Omron CX-Programmer project NewProject (CX-Programmer 9.73)

# PLC NewPLC1: CP1E E30

## Global symbols (name address type ; comment)
0.00 BOOL  ; A
0.01 BOOL  ; B
0.02 BOOL  ; C
0.03 BOOL  ; D
0.04 BOOL  ; E
0.05 BOOL  ; F
100.00 BOOL  ; G1 naik
100.01 BOOL  ; G1 turun
100.02 BOOL  ; G2 naik
100.03 BOOL  ; G2 turun
100.04 BOOL  ; G3 naik
100.05 BOOL  ; G3 turun
100.06 BOOL  ; V1 penuh
100.07 BOOL  ; V2 penuh
10.00 BOOL  ; set G1 turun
10.01 BOOL  ; set G2 turun
10.02 BOOL  ; set G3 turun
11.00 BOOL  ; NOP
D1 CHANNEL  ; data V1
D2 CHANNEL  ; data V2
T000 BOOL  ; delay G1 naik
T001 BOOL  ; delay set G1 turun
T002 BOOL  ; delay G1 turun
T004 BOOL  ; delay G2 naik
T005 BOOL  ; delay set G2 turun
T006 BOOL  ; delay G2 turun
T007 BOOL  ; delay G3 naik
T008 BOOL  ; delay set G3 turun
T009 BOOL  ; delay G3 turun
W0.01 BOOL  ; M.V1
W0.02 BOOL  ; M.V2

## Program NewProgram1 (cyclic task 0)

### Section PROGRAM

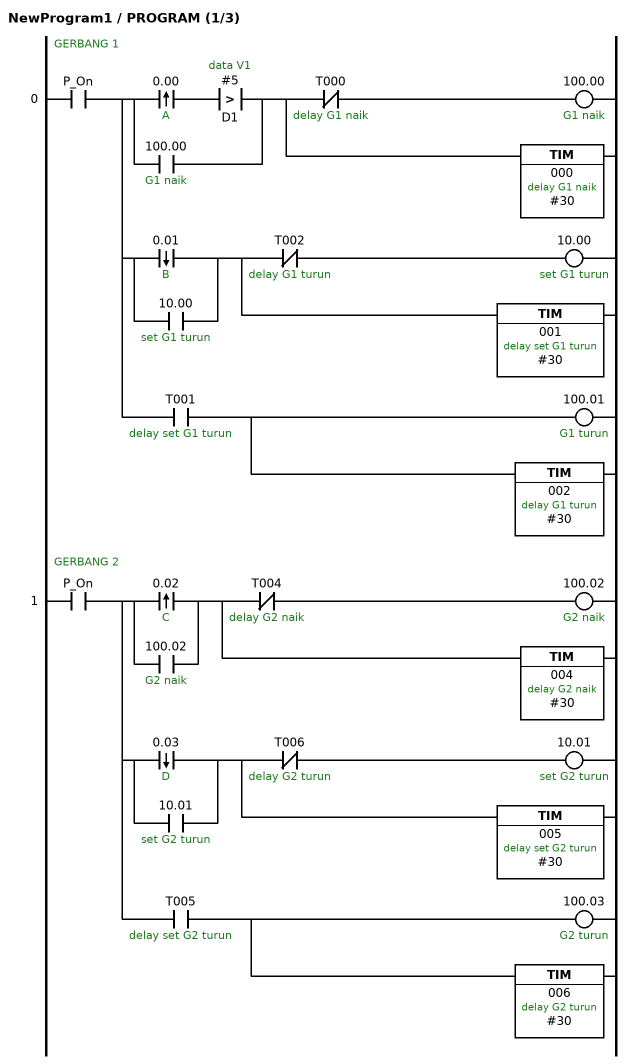
; rung 0: GERBANG 1
LD P_On
OUT TR0
@LD 0.00  ; A
AND>(320) #5 D1  ; data V1
OR 100.00  ; G1 naik
ANDLD
OUT TR1
ANDNOT T000  ; delay G1 naik
OUT 100.00  ; G1 naik
LD TR1
TIM 000 #30  ; delay G1 naik
LD TR0
%LD 0.01  ; B
OR 10.00  ; set G1 turun
ANDLD
OUT TR1
ANDNOT T002  ; delay G1 turun
OUT 10.00  ; set G1 turun
LD TR1
TIM 001 #30  ; delay set G1 turun
LD TR0
AND T001  ; delay set G1 turun
OUT 100.01  ; G1 turun
TIM 002 #30  ; delay G1 turun
; rung 1: GERBANG 2
LD P_On
OUT TR0
@LD 0.02  ; C
OR 100.02  ; G2 naik
ANDLD
OUT TR1
ANDNOT T004  ; delay G2 naik
OUT 100.02  ; G2 naik
LD TR1
TIM 004 #30  ; delay G2 naik
LD TR0
%LD 0.03  ; D
OR 10.01  ; set G2 turun
ANDLD
OUT TR1
ANDNOT T006  ; delay G2 turun
OUT 10.01  ; set G2 turun
LD TR1
TIM 005 #30  ; delay set G2 turun
LD TR0
AND T005  ; delay set G2 turun
OUT 100.03  ; G2 turun
TIM 006 #30  ; delay G2 turun

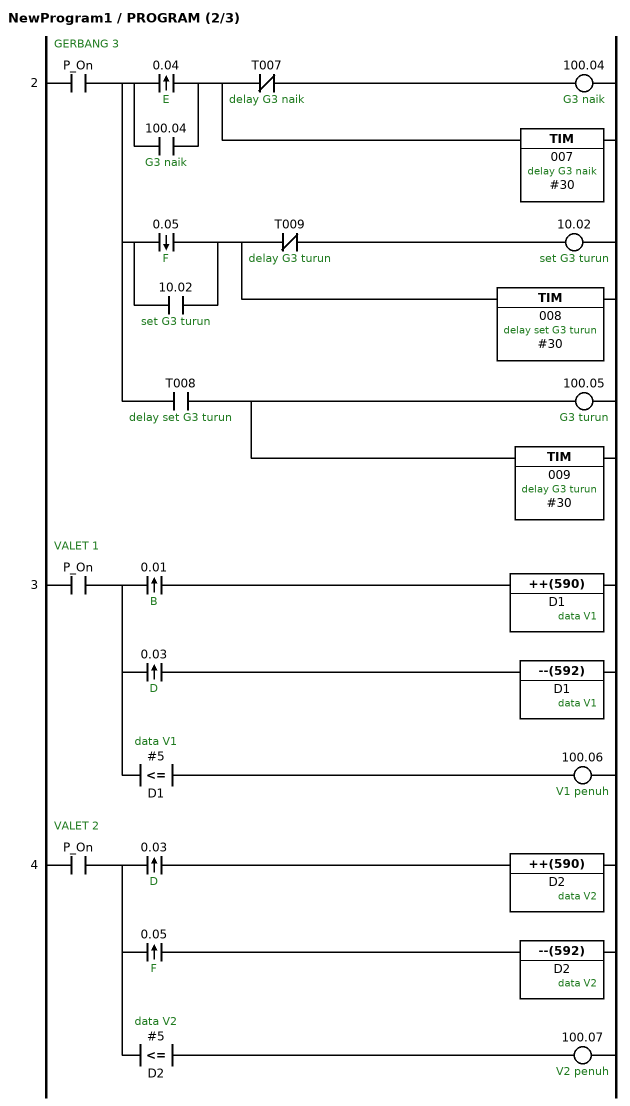
; rung 2: GERBANG 3
LD P_On
OUT TR0
@LD 0.04  ; E
OR 100.04  ; G3 naik
ANDLD
OUT TR1
ANDNOT T007  ; delay G3 naik
OUT 100.04  ; G3 naik
LD TR1
TIM 007 #30  ; delay G3 naik
LD TR0
%LD 0.05  ; F
OR 10.02  ; set G3 turun
ANDLD
OUT TR1
ANDNOT T009  ; delay G3 turun
OUT 10.02  ; set G3 turun
LD TR1
TIM 008 #30  ; delay set G3 turun
LD TR0
AND T008  ; delay set G3 turun
OUT 100.05  ; G3 turun
TIM 009 #30  ; delay G3 turun
; rung 3: VALET 1
LD P_On
OUT TR0
@AND 0.01  ; B
++(590) D1  ; data V1
LD TR0
@AND 0.03  ; D
--(592) D1  ; data V1
LD TR0
AND<=(315) #5 D1  ; data V1
OUT 100.06  ; V1 penuh
; rung 4: VALET 2
LD P_On
OUT TR0
@AND 0.03  ; D
++(590) D2  ; data V2
LD TR0
@AND 0.05  ; F
--(592) D2  ; data V2
LD TR0
AND<=(315) #5 D2  ; data V2
OUT 100.07  ; V2 penuh

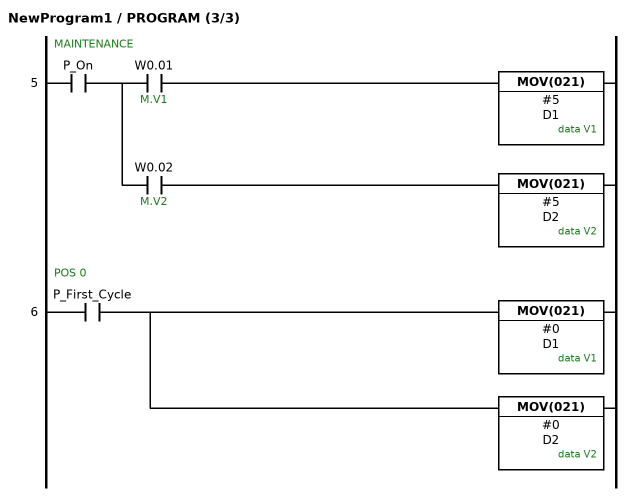
; rung 5: MAINTENANCE
LD P_On
OUT TR0
AND W0.01  ; M.V1
MOV(021) #5 D1  ; data V1
LD TR0
AND W0.02  ; M.V2
MOV(021) #5 D2  ; data V2
; rung 6: POS 0
LD P_First_Cycle
MOV(021) #0 D1  ; data V1
MOV(021) #0 D2  ; data V2

### Section IN_OUT

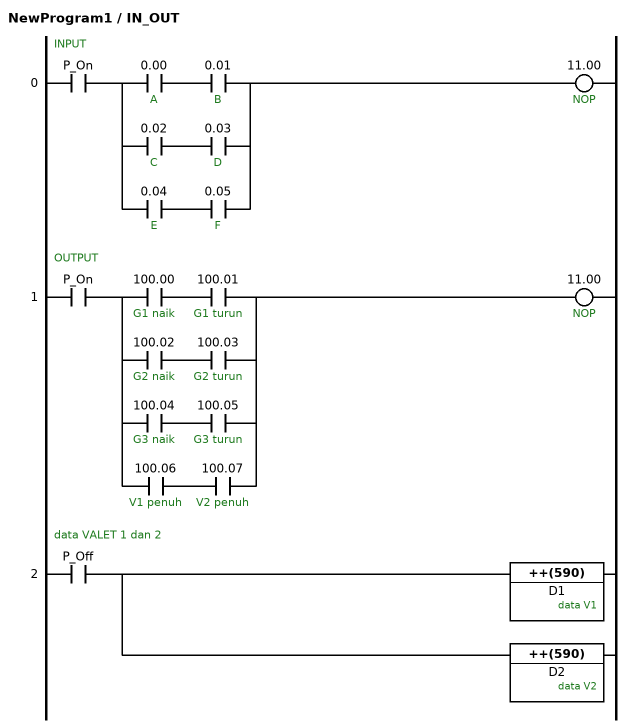
; rung 0: INPUT
LD P_On
LD 0.00  ; A
AND 0.01  ; B
LD 0.02  ; C
AND 0.03  ; D
ORLD
LD 0.04  ; E
AND 0.05  ; F
ORLD
ANDLD
OUT 11.00  ; NOP
; rung 1: OUTPUT
LD P_On
LD 100.00  ; G1 naik
AND 100.01  ; G1 turun
LD 100.02  ; G2 naik
AND 100.03  ; G2 turun
ORLD
LD 100.04  ; G3 naik
AND 100.05  ; G3 turun
ORLD
LD 100.06  ; V1 penuh
AND 100.07  ; V2 penuh
ORLD
ANDLD
OUT 11.00  ; NOP
; rung 2: data VALET 1 dan 2
LD P_Off
++(590) D1  ; data V1
++(590) D2  ; data V2

### Section END
; rung 0
END(001)